// TIA Portal V17 export
// export: Created 2025-08-05T09:36:01.8437012Z, ExportSetting WithDefaults, DisplayName Totally Integrated Automation Portal, DisplayVersion V17, DisplayName TIA Portal Openness, DisplayVersion V17, DisplayName TIA Portal Version Control Interface, DisplayVersion V17, DisplayName SINAMICS Startdrive Advanced, DisplayVersion V17, DisplayName SINAMICS Startdrive G130, G150, S120, S150, SINAMICS MV, S210, DisplayVersion V17, DisplayName SINAMICS Startdrive G110M, G120, G120C, G120D, G120P, G115D, DisplayVersion V17, DisplayName STEP 7 Professional, DisplayVersion V17, DisplayName STEP 7 Safety, DisplayVersion V17, DisplayName WinCC Advanced, DisplayVersion V17
TYPE "YLR_Inputs"
// stored: IsFailsafeCompliant false
   STRUCT
      Command_Buffer_Overflow : Bool;   // Command_Buffer_Overflow
      Overheat : Bool;   // Overheat
      Emission_On : Bool;   // Emission_On
      High_Back_Reflection : Bool;   // High_Back_Reflection
      Analogue_Power_Control_Enabled : Bool;   // Analogue_Power_Control_Enabled
      Pulse_Too_Long : Bool;   // Pulse_Too_Long
      Reserved_1 : Bool;   // Reserved_1
      Reserved_2 : Bool;   // Reserved_2
      Aiming_Beam_On : Bool;   // Aiming_Beam_On
      Pulse_Too_Short : Bool;   // Pulse_Too_Short
      Pulsed_Mode : Bool;   // Pulsed_Mode
      Power_Supply_Off : Bool;   // Power_Supply_Off
      Modulation_Enabled : Bool;   // Modulation_Enabled
      Reserved_3 : Bool;   // Reserved_3
      Reserved_4 : Bool;   // Reserved_4
      Emission_Starting : Bool;   // Emission_Starting
      Gate_Mode_Enabled : Bool;   // Gate_Mode_Enabled
      High_Pulse_Energy : Bool;   // High_Pulse_Energy
      Hardware_Emission_Control_Enabled : Bool;   // Hardware_Emission_Control_Enabled
      Power_Supply_Failure : Bool;   // Power_Supply_Failure
      Front_Panel_Display_Locked : Bool;   // Front_Panel_Display_Locked
      Keyswitch_in_REM_Position : Bool;   // Keyswitch_in_REM_Position
      Waveform_Mode_On : Bool;   // Waveform_Mode_On
      Duty_Cycle_Too_High : Bool;   // Duty_Cycle_Too_High
      Low_Temperature : Bool;   // Low_Temperature
      Power_Supply_Alarm : Bool;   // Power_Supply_Alarm
      Reserved_5 : Bool;   // Reserved_5
      Hardware_Aiming_Beam_Control_Enabled : Bool;   // Hardware_Aiming_Beam_Control_Enabled
      Aiming_Beam_Alarm : Bool;   // Aiming_Beam_Alarm
      Critical_Error : Bool;   // Critical_Error
      Fiberlock_Interlock_Active : Bool;   // Fiberlock_Interlock_Active
      High_Average_Power : Bool;   // High_Average_Power
   END_STRUCT;
END_TYPE
